{attribute addProperty BoxType "EPP1518-0002-0016"}
{attribute addProperty Id "ControlAT %Q*Control_051AC2241620Set_counter_valueAT %Q*UDINT32417"}
{attribute addProperty CRC "3342441697"}
{attribute addProperty SizeInBites "48"}
{attribute addProperty SizeInBytes "6"}
TYPE CNT_Output_Channel_C7399CE1 :
STRUCT
	{attribute addProperty Name "Control"}
	Control AT %Q* : Control_051AC224;
	{attribute addProperty Name "Set_counter_value"}
	Set_counter_value AT %Q* : UDINT;
END_STRUCT
END_TYPE

(* stored: Version 1.2.0.0, ProductVersion 3.1.4024.9
   DUT CNT_Output_Channel_C7399CE1: Id {d08d8315-1e39-4a10-8b63-0560cb9e2b45} *)
